(* PLC project  *)

PROGRAM P

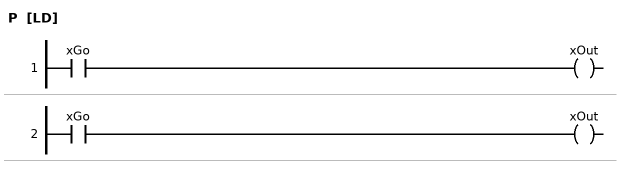
(* LD diagram, written out as Structured Text *)
xOut := xGo;
xOut := xGo;
END_PROGRAM
